{attribute addProperty BoxType "EL2521-0124-0018"}
{attribute addProperty Id "StatusAT %I*Status_8A45CCAE162"}
{attribute addProperty CRC "2787335905"}
{attribute addProperty SizeInBites "16"}
{attribute addProperty SizeInBytes "2"}
TYPE PLS_Status_A6235EE1 :
STRUCT
	{attribute addProperty Name "Status"}
	Status AT %I* : Status_8A45CCAE;
END_STRUCT
END_TYPE

(* stored: Version 1.2.0.0, ProductVersion 3.1.4024.9
   DUT PLS_Status_A6235EE1: Id {b426e2c4-3dfb-432b-a39e-0d21a7cc19ba} *)
